PROGRAM Status_and_Alarms
VAR

END_VAR

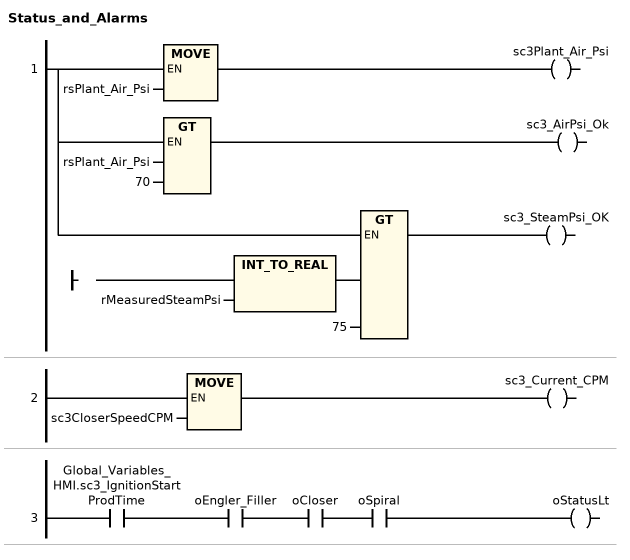
// NETWORK 1
sc3Plant_Air_Psi := rsPlant_Air_Psi;
sc3_AirPsi_Ok := rsPlant_Air_Psi > 70;
sc3_SteamPsi_OK := INT_TO_REAL(rMeasuredSteamPsi) > 75;

// NETWORK 2
sc3_Current_CPM := sc3CloserSpeedCPM;

// NETWORK 3
oStatusLt := Global_Variables_HMI.sc3_IgnitionStartProdTime AND oEngler_Filler AND oCloser AND oSpiral;

END_PROGRAM

(* stored: Version 1.1.0.1, ProductVersion 3.1.4024.15
   POU Status_and_Alarms: Id {9e85b3c3-8b0c-4813-8371-80c58ded9680}, SpecialFunc None *)
